FUNCTION_BLOCK FB_LineAxis
VAR_INPUT
	System:					REFERENCE TO ST_System;
END_VAR
VAR_OUTPUT
	Moving:					BOOL;
END_VAR
VAR
	_moving:				BOOL;
END_VAR

Moving:=FALSE;

IF System.stInput.bReset THEN
	Moving:=_moving:=FALSE;
END_IF


IF System.stMode.stDeviceEnable.bAuto OR System.stMode.stDeviceEnable.bManual THEN
	Moving:=_moving;
END_IF

METHOD M_Jog : BOOL
VAR_INPUT
	Command:				INT;// -1:反转 0:停止 1:正转
END_VAR
M_Jog:=FALSE;
IF Command=1 THEN
	_moving:=TRUE;
	M_Jog:=TRUE;
END_IF

IF Command=0 THEN
	_moving:=FALSE;
	M_Jog:=TRUE;
END_IF
END_METHOD

END_FUNCTION_BLOCK

(* stored: Version 1.1.0.1, ProductVersion 3.1.4024.3
   POU FB_LineAxis: Id {b1eab20f-524e-4969-82ec-b988eb20465a}, SpecialFunc None
   Method M_Jog: Id {5bca00aa-b573-4724-a945-d56bf73ef527} *)
